// Mitsubishi GX Works2 project: ServMotor4   PLC: Q03UDV

PROGRAM MAIN
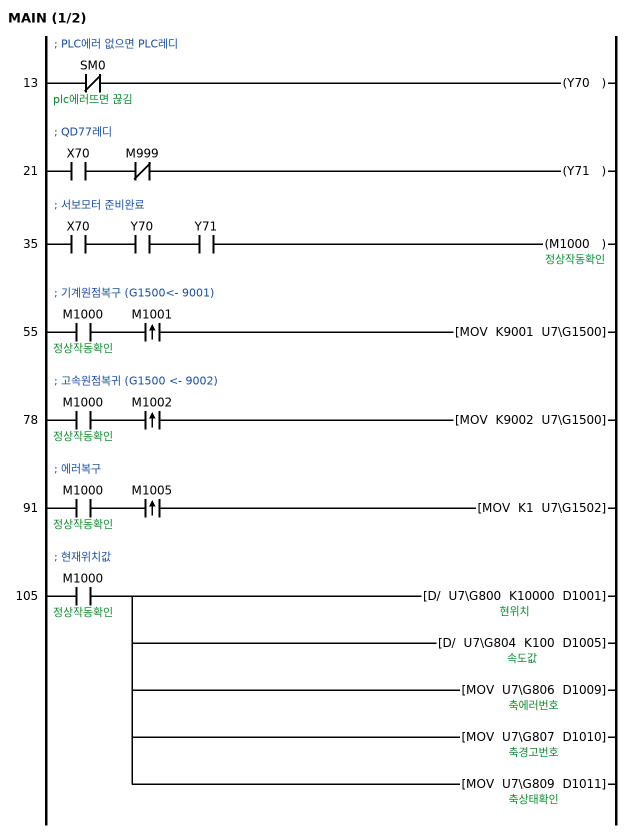
; PLC에러 없으면 PLC레디
13    LDI     SM0  ; plc에러뜨면 끊김
      OUT     Y70
; QD77레디
21    LD      X70
      ANI     M999
      OUT     Y71
; 서보모터 준비완료
35    LD      X70
      AND     Y70
      AND     Y71
      OUT     M1000  ; 정상작동확인
; 기계원점복구 (G1500<- 9001)
55    LD      M1000  ; 정상작동확인
      ANDP    M1001
      MOV     K9001 U7\G1500
; 고속원점복귀 (G1500 <- 9002)
78    LD      M1000  ; 정상작동확인
      ANDP    M1002
      MOV     K9002 U7\G1500
; 에러복구
91    LD      M1000  ; 정상작동확인
      ANDP    M1005
      MOV     K1 U7\G1502
; 현재위치값
105   LD      M1000  ; 정상작동확인
      D/      U7\G800 K10000 D1001  ; 현위치
      D/      U7\G804 K100 D1005  ; 속도값
      MOV     U7\G806 D1009  ; 축에러번호
      MOV     U7\G807 D1010  ; 축경고번호
      MOV     U7\G809 D1011  ; 축상태확인
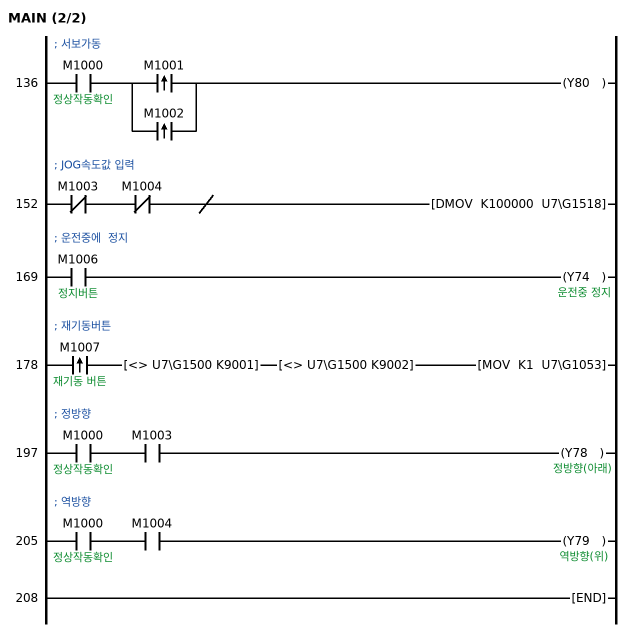
; 서보가동
136   LD      M1000  ; 정상작동확인
      LDP     M1001
      ORP     M1002
      ANB
      OUT     Y80
; JOG속도값 입력
152   LDI     M1003
      ANI     M1004
      INV
      DMOV    K100000 U7\G1518
; 운전중에  정지
169   LD      M1006  ; 정지버튼
      OUT     Y74  ; 운전중 정지
; 재기동버튼
178   LDP     M1007  ; 재기동 버튼
      AND<>   U7\G1500 K9001
      AND<>   U7\G1500 K9002
      MOV     K1 U7\G1053
; 정방향
197   LD      M1000  ; 정상작동확인
      AND     M1003
      OUT     Y78  ; 정방향(아래)
; 역방향
205   LD      M1000  ; 정상작동확인
      AND     M1004
      OUT     Y79  ; 역방향(위)
208   END
END_PROGRAM

// device comments not shown above
D1000  ; d1000~d1003
D1012  ; 에러메세지
